Staubli VAL3: IOModule.dtx

public num BASIC_IN
public num BASIC_IN_2
public num BASIC_OUT
public num BASIC_OUT_2
public num UNKNOWN
public num USER_IN
public num VALVE_OUT
